(*******************************************************************************
                          protoc-gen-twincat v0.0.0.0                           
             https://github.bhs-world.com/CorrML/protoc-gen-twincat             
*******************************************************************************)
{attribute 'no-analysis'}
TYPE ST_Foo :
STRUCT
	bar : ST_Bar;
	baz : ARRAY[0..2] OF ST_Baz;
	baz_count : UDINT; // Implict generated field for actual number of items in array baz
END_STRUCT
END_TYPE

(* stored: Version 1.1.0.1
   DUT ST_Foo: Id {52ee6fce-0584-4435-ada8-b7d6f1aca3da} *)
